PROGRAM AgitationMechanismCtrl
VAR

	fbV2StnAgitationCtrl1: fbV2_AgitationMechanismCtrl;
	fbV2StnAgitationCtrl2: fbV2_AgitationMechanismCtrl;

	iStnAgitation1DelayOffTimerEV: INT;
	iStnAgitation2DelayOffTimerEV: INT;
  btestVSCode : INT;

END_VAR

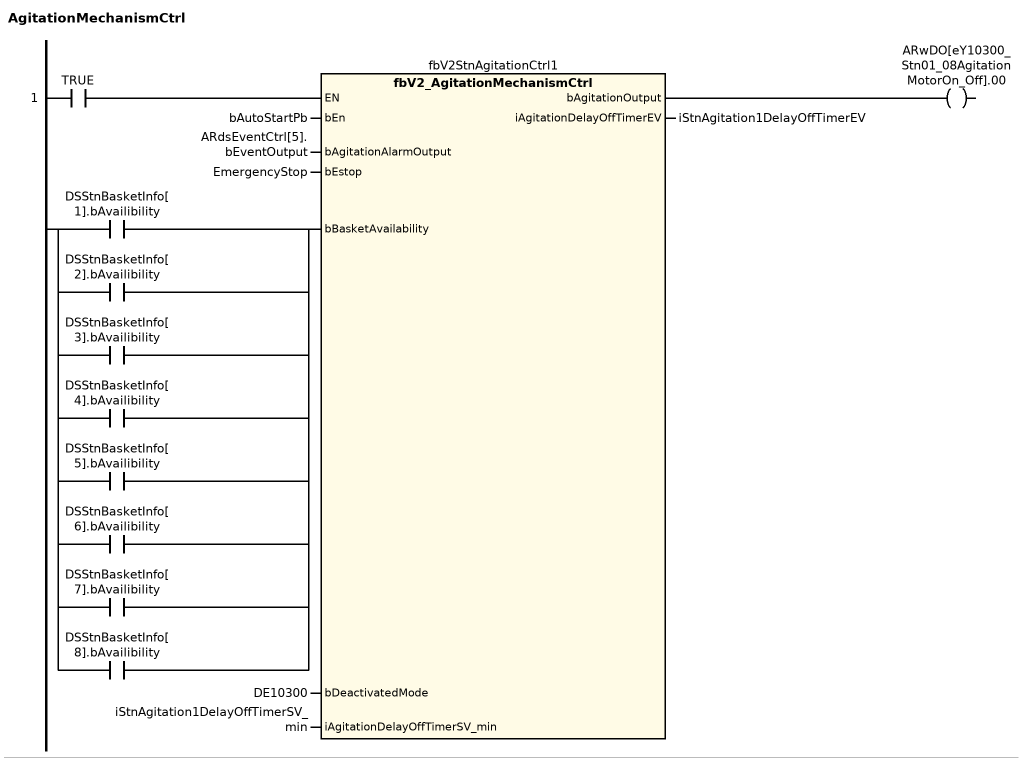
// NETWORK 1
fbV2StnAgitationCtrl1(
    bEn := bAutoStartPb,
    bAgitationAlarmOutput := ARdsEventCtrl[5].bEventOutput,
    bEstop := EmergencyStop,
    bBasketAvailability := DSStnBasketInfo[1].bAvailibility OR DSStnBasketInfo[2].bAvailibility OR DSStnBasketInfo[3].bAvailibility OR DSStnBasketInfo[4].bAvailibility OR DSStnBasketInfo[5].bAvailibility OR DSStnBasketInfo[6].bAvailibility OR DSStnBasketInfo[7].bAvailibility OR DSStnBasketInfo[8].bAvailibility,
    bDeactivatedMode := DE10300,
    iAgitationDelayOffTimerSV_min := iStnAgitation1DelayOffTimerSV_min,
    iAgitationDelayOffTimerEV => iStnAgitation1DelayOffTimerEV); // fbV2_AgitationMechanismCtrl
ARwDO[eY10300_Stn01_08AgitationMotorOn_Off].00 := fbV2StnAgitationCtrl1.bAgitationOutput;

END_PROGRAM

(* stored: Version 1.1.0.1, ProductVersion 3.1.4024.12
   POU AgitationMechanismCtrl: Id {570547af-8638-48a5-b40c-7c158b69612b}, SpecialFunc None *)
